ABB RAPID module: 00064353

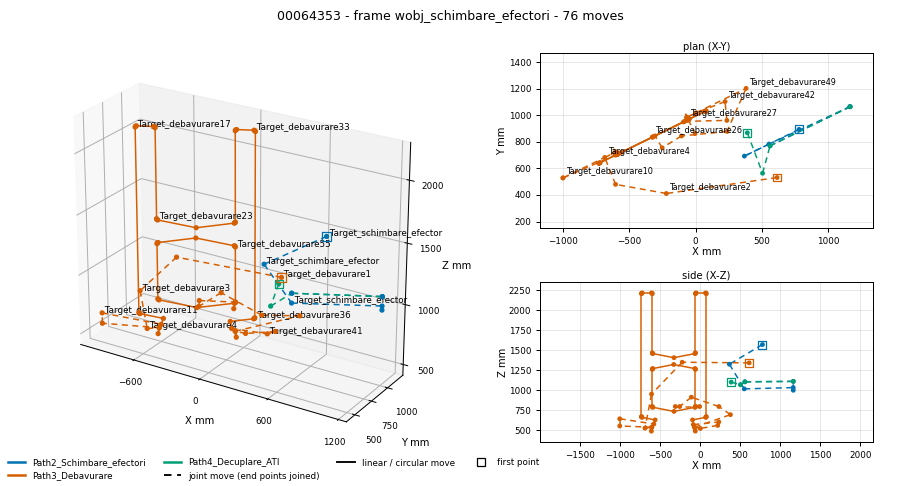
[picture p0: tool path of 00064353 in frame wobj_schimbare_efectori, 76 of 136 moves have a stored position in this frame; points joined in program order, loops and branches not executed]
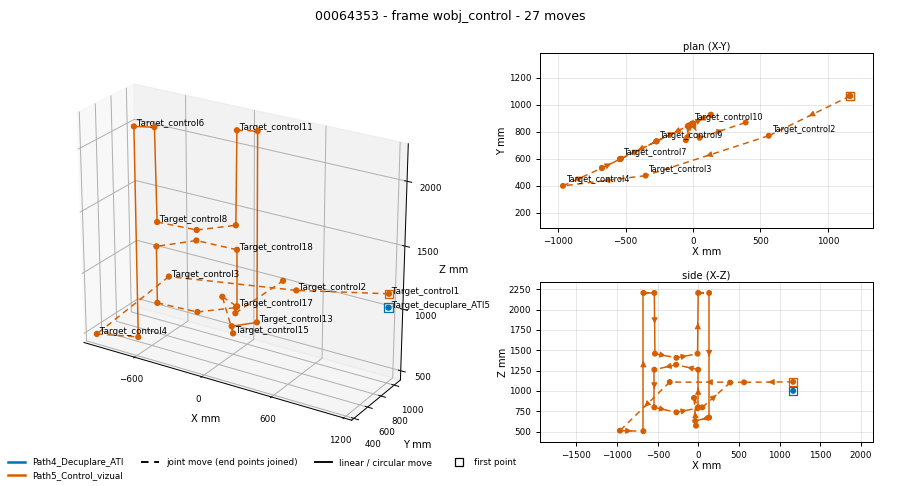
[picture p1: tool path of 00064353 in frame wobj_control, 27 of 136 moves have a stored position in this frame; points joined in program order, loops and branches not executed]
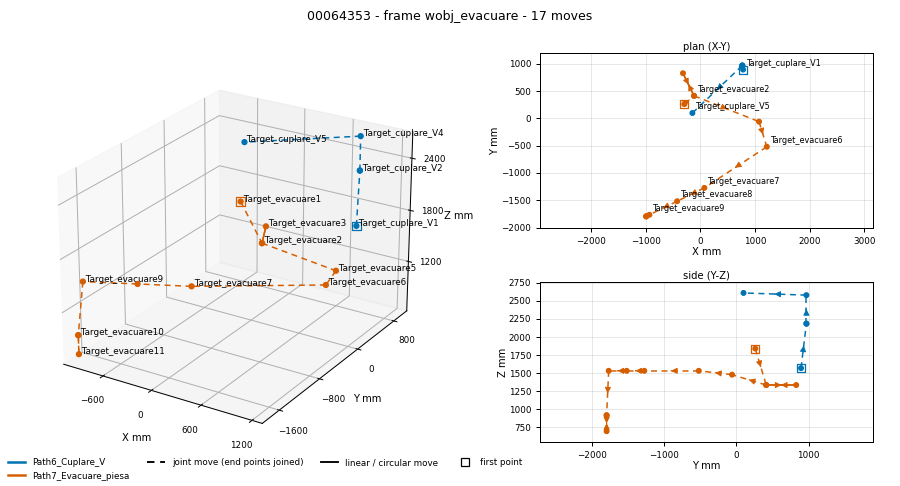
[picture p2: tool path of 00064353 in frame wobj_evacuare, 17 of 136 moves have a stored position in this frame; points joined in program order, loops and branches not executed]
MODULE Module1
	CONST robtarget Target_20_2:=[[0,0.000001,500],[0,0,1,-0.000000001],[-2,-1,0,0],[9E+09,9E+09,9E+09,9E+09,9E+09,9E+09]];
	CONST robtarget Target_10:=[[3.472963553,17.439983187,29.999999981],[0,0,1,-0.000000001],[0,-1,0,0],[9E+09,9E+09,9E+09,9E+09,9E+09,9E+09]];
	CONST robtarget Target_20:=[[0,0.000001,500],[0,0,1,-0.000000001],[-2,-1,0,0],[9E+09,9E+09,9E+09,9E+09,9E+09,9E+09]];
	CONST robtarget Target_20_2_3:=[[493.307337926,-365.839908027,1036.754553389],[0,0,1,-0.000000001],[-1,0,0,0],[9E+09,9E+09,9E+09,9E+09,9E+09,9E+09]];
	CONST robtarget Target_30:=[[-807.278732186,-859.510215676,1233.208067661],[0.579227966,0.405579787,-0.5,-0.5],[0,0,0,0],[9E+09,9E+09,9E+09,9E+09,9E+09,9E+09]];
	CONST robtarget Target_30_3:=[[-1171.792571204,-860.224752875,1298.599208728],[0.579227966,0.405579787,-0.5,-0.5],[1,0,0,0],[9E+09,9E+09,9E+09,9E+09,9E+09,9E+09]];
	CONST robtarget Target_70:=[[-584.684106736,-1037.65235773,1745.210003217],[0.579227966,0.405579787,-0.5,-0.5],[0,0,0,4],[9E+09,9E+09,9E+09,9E+09,9E+09,9E+09]];
	CONST robtarget Target_120:=[[614.35326876,531.541624289,1341.660223262],[0.630196274,-0.425266678,-0.564932078,-0.320706495],[0,0,1,0],[9E+09,9E+09,9E+09,9E+09,9E+09,9E+09]];
	CONST robtarget Target_130:=[[-220.756964436,411.144811502,1349.578986688],[0.630196274,-0.425266678,-0.564932078,-0.320706495],[1,1,0,1],[9E+09,9E+09,9E+09,9E+09,9E+09,9E+09]];
	CONST robtarget Target_140:=[[-603.640790819,480.038707024,951.826023694],[0.630196274,-0.425266678,-0.564932078,-0.320706495],[1,0,1,1],[9E+09,9E+09,9E+09,9E+09,9E+09,9E+09]];
	CONST robtarget Target_150:=[[-684.956865831,682.802213826,527.356838346],[0.630196274,-0.425266678,-0.564932078,-0.320706495],[1,0,1,1],[9E+09,9E+09,9E+09,9E+09,9E+09,9E+09]];
	CONST robtarget Target_160:=[[-600.231193595,724.230019574,538.596152517],[0.630196274,-0.425266678,-0.564932078,-0.320706495],[1,0,1,1],[9E+09,9E+09,9E+09,9E+09,9E+09,9E+09]];
	CONST robtarget Target_170:=[[-615.502782618,744.38841834,511.008322261],[0.630196274,-0.425266678,-0.564932078,-0.320706495],[1,0,1,1],[9E+09,9E+09,9E+09,9E+09,9E+09,9E+09]];
	CONST robtarget Target_180:=[[-605.289704553,715.096779867,490.071182954],[0.630196274,-0.425266678,-0.564932078,-0.320706495],[1,0,1,1],[9E+09,9E+09,9E+09,9E+09,9E+09,9E+09]];
	CONST robtarget Target_190:=[[-592.759513668,700.25774586,516.943595123],[0.630196274,-0.425266678,-0.564932078,-0.320706495],[1,0,1,1],[9E+09,9E+09,9E+09,9E+09,9E+09,9E+09]];
	CONST robtarget Target_200:=[[-600.231193595,724.230019574,538.596152517],[0.630196274,-0.425266678,-0.564932078,-0.320706495],[1,0,1,1],[9E+09,9E+09,9E+09,9E+09,9E+09,9E+09]];
	CONST robtarget Target_210:=[[-1000.069986007,528.723234139,554.74513186],[0.630196274,-0.425266678,-0.564932078,-0.320706495],[1,0,1,1],[9E+09,9E+09,9E+09,9E+09,9E+09,9E+09]];
	CONST robtarget Target_210_2:=[[-1000.069986007,528.723234139,644.473462045],[0.74632501,0.144907108,-0.626241041,0.172693565],[1,-1,2,1],[9E+09,9E+09,9E+09,9E+09,9E+09,9E+09]];
	CONST robtarget Target_220:=[[-574.244255672,714.673851005,578.901883612],[0.74632501,0.144907108,-0.626241041,0.172693565],[1,-2,-2,1],[9E+09,9E+09,9E+09,9E+09,9E+09,9E+09]];
	CONST robtarget Target_230:=[[-558.661492442,722.293261641,630.386873665],[0.74632501,0.144907108,-0.626241041,0.172693565],[1,-2,-2,1],[9E+09,9E+09,9E+09,9E+09,9E+09,9E+09]];
	CONST robtarget Target_240:=[[-721.925864829,642.46285692,662.431918782],[0.74632501,0.144907108,-0.626241041,0.172693565],[1,-1,-2,1],[9E+09,9E+09,9E+09,9E+09,9E+09,9E+09]];
	CONST robtarget Target_250:=[[-727.247702444,639.860669777,665.852120215],[0.74632501,0.144907108,-0.626241041,0.172693565],[1,-1,-2,1],[9E+09,9E+09,9E+09,9E+09,9E+09,9E+09]];
	CONST robtarget Target_260:=[[-729.349460263,638.832985813,672.279996312],[0.74632501,0.144907108,-0.626241041,0.172693565],[1,-1,-2,1],[9E+09,9E+09,9E+09,9E+09,9E+09,9E+09]];
	CONST robtarget Target_270:=[[-729.349460263,638.832985813,2203.889],[0.74632501,0.144907108,-0.626241041,0.172693565],[1,-1,-1,1],[9E+09,9E+09,9E+09,9E+09,9E+09,9E+09]];
	CONST robtarget Target_280:=[[-726.718231405,640.119562068,2210.960067812],[0.74632501,0.144907108,-0.626241041,0.172693565],[1,-1,-1,1],[9E+09,9E+09,9E+09,9E+09,9E+09,9E+09]];
	CONST robtarget Target_290:=[[-720.36588301,643.22563191,2213.889],[0.970550763,-0.019647992,0.084912189,0.22457759],[1,0,-2,1],[9E+09,9E+09,9E+09,9E+09,9E+09,9E+09]];
	CONST robtarget Target_300:=[[-603.579378711,700.33003116,2213.889],[0.970550763,-0.019647992,0.084912189,0.22457759],[1,0,-2,1],[9E+09,9E+09,9E+09,9E+09,9E+09,9E+09]];
	CONST robtarget Target_310:=[[-597.227030315,703.436101002,2210.960067812],[0.970550763,-0.019647992,0.084912189,0.22457759],[1,0,-2,1],[9E+09,9E+09,9E+09,9E+09,9E+09,9E+09]];
	CONST robtarget Target_320:=[[-594.595801457,704.722677256,2203.889],[0.970550763,-0.019647992,0.084912189,0.22457759],[1,0,-2,1],[9E+09,9E+09,9E+09,9E+09,9E+09,9E+09]];
	CONST robtarget Target_330:=[[-594.595801457,704.722677256,1467.279996312],[0.970550763,-0.019647992,0.084912189,0.22457759],[1,0,-2,1],[9E+09,9E+09,9E+09,9E+09,9E+09,9E+09]];
	CONST robtarget Target_340:=[[-592.494043638,705.75036122,1460.852120215],[0.970550763,-0.019647992,0.084912189,0.22457759],[1,0,-2,1],[9E+09,9E+09,9E+09,9E+09,9E+09,9E+09]];
	CONST robtarget Target_350:=[[-587.172206023,708.352548362,1457.431918782],[0.970550763,-0.019647992,0.084912189,0.22457759],[1,0,-2,1],[9E+09,9E+09,9E+09,9E+09,9E+09,9E+09]];
	CONST robtarget Target_360:=[[-323.528502026,837.264835131,1406.297094376],[0.970550763,-0.019647992,0.084912189,0.22457759],[1,0,-1,1],[9E+09,9E+09,9E+09,9E+09,9E+09,9E+09]];
	CONST robtarget Target_370:=[[-63.004761668,964.65157192,1457.431918782],[0.970550763,-0.019647992,0.084912189,0.22457759],[1,0,-1,1],[9E+09,9E+09,9E+09,9E+09,9E+09,9E+09]];
	CONST robtarget Target_380:=[[-57.682924053,967.253759063,1460.852120215],[0.970550763,-0.019647992,0.084912189,0.22457759],[1,0,-1,1],[9E+09,9E+09,9E+09,9E+09,9E+09,9E+09]];
	CONST robtarget Target_390:=[[-55.581166233,968.281443027,1467.279996312],[0.970550763,-0.019647992,0.084912189,0.22457759],[1,0,-1,1],[9E+09,9E+09,9E+09,9E+09,9E+09,9E+09]];
	CONST robtarget Target_400:=[[-55.581166233,968.281443027,2203.889],[0.970550763,-0.019647992,0.084912189,0.22457759],[1,0,-1,1],[9E+09,9E+09,9E+09,9E+09,9E+09,9E+09]];
	CONST robtarget Target_410:=[[-52.949937375,969.568019281,2210.960067812],[0.970550763,-0.019647992,0.084912189,0.22457759],[1,0,-1,1],[9E+09,9E+09,9E+09,9E+09,9E+09,9E+09]];
	CONST robtarget Target_420:=[[-46.59758898,972.674089123,2213.889],[0.970550763,-0.019647992,0.084912189,0.22457759],[1,0,-1,1],[9E+09,9E+09,9E+09,9E+09,9E+09,9E+09]];
	CONST robtarget Target_430:=[[70.188915319,1029.778488373,2213.889],[0.970550763,-0.019647992,0.084912189,0.22457759],[0,0,-1,1],[9E+09,9E+09,9E+09,9E+09,9E+09,9E+09]];
	CONST robtarget Target_440:=[[76.541263714,1032.884558215,2210.960067812],[0.970550763,-0.019647992,0.084912189,0.22457759],[0,0,-1,1],[9E+09,9E+09,9E+09,9E+09,9E+09,9E+09]];
	CONST robtarget Target_450:=[[79.172492573,1034.171134469,2203.889],[0.626241041,-0.172693565,0.74632501,0.144907108],[1,1,-2,1],[9E+09,9E+09,9E+09,9E+09,9E+09,9E+09]];
	CONST robtarget Target_460:=[[79.172492573,1034.171134469,672.279996312],[0.626241041,-0.172693565,0.74632501,0.144907108],[1,0,-1,1],[9E+09,9E+09,9E+09,9E+09,9E+09,9E+09]];
	CONST robtarget Target_470:=[[77.070734753,1033.143450506,665.852120215],[0.626241041,-0.172693565,0.74632501,0.144907108],[1,0,-1,1],[9E+09,9E+09,9E+09,9E+09,9E+09,9E+09]];
	CONST robtarget Target_480:=[[71.748897138,1030.541263363,662.431918782],[0.626241041,-0.172693565,0.74632501,0.144907108],[1,0,-1,1],[9E+09,9E+09,9E+09,9E+09,9E+09,9E+09]];
	CONST robtarget Target_490:=[[-91.515475248,950.710858642,630.386873665],[0.626241041,-0.172693565,0.74632501,0.144907108],[1,1,-1,1],[9E+09,9E+09,9E+09,9E+09,9E+09,9E+09]];
	CONST robtarget Target_500:=[[-82.17325952,955.27886605,571.409990938],[0.626241041,-0.172693565,0.74632501,0.144907108],[1,1,-1,1],[9E+09,9E+09,9E+09,9E+09,9E+09,9E+09]];
	CONST robtarget Target_500_2:=[[235.647161917,962.336296138,604.766182313],[0.626241041,-0.172693565,0.74632501,0.144907108],[0,0,-1,1],[9E+09,9E+09,9E+09,9E+09,9E+09,9E+09]];
	CONST robtarget Target_500_2_2:=[[222.398190082,1104.203348059,561.899220237],[0.320706496,-0.564932078,0.425266677,0.630196274],[0,1,-2,0],[9E+09,9E+09,9E+09,9E+09,9E+09,9E+09]];
	CONST robtarget Target_510:=[[4.592265391,1019.966932715,523.466438018],[0.425266678,-0.630196274,0.320706495,0.564932078],[0,1,-2,0],[9E+09,9E+09,9E+09,9E+09,9E+09,9E+09]];
	CONST robtarget Target_520:=[[-67.51635848,984.708409724,538.596152517],[0.425266678,-0.630196274,0.320706495,0.564932078],[0,1,-2,0],[9E+09,9E+09,9E+09,9E+09,9E+09,9E+09]];
	CONST robtarget Target_530:=[[-74.04786326,1009.140395264,511.008322261],[0.425266678,-0.630196274,0.320706495,0.564932078],[0,1,-2,0],[9E+09,9E+09,9E+09,9E+09,9E+09,9E+09]];
	CONST robtarget Target_540:=[[-57.20170243,983.09209564,490.071182954],[0.425266678,-0.630196274,0.320706495,0.564932078],[0,1,-2,0],[9E+09,9E+09,9E+09,9E+09,9E+09,9E+09]];
	CONST robtarget Target_550:=[[-53.184944606,964.090299134,516.943595123],[0.425266678,-0.630196274,0.320706495,0.564932078],[0,1,-2,0],[9E+09,9E+09,9E+09,9E+09,9E+09,9E+09]];
	CONST robtarget Target_560:=[[-67.51635848,984.708409724,538.596152517],[0.425266678,-0.630196274,0.320706495,0.564932078],[0,1,-2,0],[9E+09,9E+09,9E+09,9E+09,9E+09,9E+09]];
	CONST robtarget Target_570:=[[380.563228786,1203.803208398,695.774665043],[0.425266678,-0.630196274,0.320706495,0.564932078],[0,1,-2,0],[9E+09,9E+09,9E+09,9E+09,9E+09,9E+09]];
	CONST robtarget Target_580_3:=[[236.855316057,878.977367128,797.279996312],[0.626241041,-0.172693565,0.74632501,0.144907108],[0,0,-1,1],[9E+09,9E+09,9E+09,9E+09,9E+09,9E+09]];
	CONST robtarget Target_740:=[[-106.574951523,844.917671275,913.754533399],[0.626241041,-0.172693565,0.74632501,0.144907108],[1,1,-1,1],[9E+09,9E+09,9E+09,9E+09,9E+09,9E+09]];
	CONST robtarget Target_580_3_2:=[[-251.957733199,755.881530829,797.279996312],[0.626241041,-0.172693565,0.74632501,0.144907108],[1,1,-1,1],[9E+09,9E+09,9E+09,9E+09,9E+09,9E+09]];
	CONST robtarget Target_580:=[[-306.602704629,845.540941159,797.279996312],[0.626241041,-0.172693565,0.74632501,0.144907108],[1,1,-1,1],[9E+09,9E+09,9E+09,9E+09,9E+09,9E+09]];
	CONST robtarget Target_590:=[[-55.581166233,968.281443027,797.279996312],[0.626241041,-0.172693565,0.74632501,0.144907108],[1,1,-1,1],[9E+09,9E+09,9E+09,9E+09,9E+09,9E+09]];
	CONST robtarget Target_600:=[[-55.581166233,968.281443027,1260.498003688],[0.626241041,-0.172693565,0.74632501,0.144907108],[1,1,-1,1],[9E+09,9E+09,9E+09,9E+09,9E+09,9E+09]];
	CONST robtarget Target_610:=[[-57.682924053,967.253759063,1266.925879785],[0.626241041,-0.172693565,0.74632501,0.144907108],[1,1,-1,1],[9E+09,9E+09,9E+09,9E+09,9E+09,9E+09]];
	CONST robtarget Target_620:=[[-63.004761668,964.65157192,1270.346081218],[0.626241041,-0.172693565,0.74632501,0.144907108],[1,1,-1,1],[9E+09,9E+09,9E+09,9E+09,9E+09,9E+09]];
	CONST robtarget Target_630:=[[-326.648465665,835.739285151,1321.480905624],[0.626241041,-0.172693565,0.74632501,0.144907108],[1,1,-1,1],[9E+09,9E+09,9E+09,9E+09,9E+09,9E+09]];
	CONST robtarget Target_640:=[[-587.172206023,708.352548362,1270.346081218],[0.626241041,-0.172693565,0.74632501,0.144907108],[1,1,-1,1],[9E+09,9E+09,9E+09,9E+09,9E+09,9E+09]];
	CONST robtarget Target_650:=[[-592.494043638,705.75036122,1266.925879785],[0.626241041,-0.172693565,0.74632501,0.144907108],[1,1,-1,1],[9E+09,9E+09,9E+09,9E+09,9E+09,9E+09]];
	CONST robtarget Target_660:=[[-594.595801457,704.722677256,1260.498003688],[0.626241041,-0.172693565,0.74632501,0.144907108],[1,1,-1,1],[9E+09,9E+09,9E+09,9E+09,9E+09,9E+09]];
	CONST robtarget Target_670:=[[-594.595801457,704.722677256,797.279996312],[0.626241041,-0.172693565,0.74632501,0.144907108],[1,1,-1,1],[9E+09,9E+09,9E+09,9E+09,9E+09,9E+09]];
	CONST robtarget Target_680:=[[-592.494043638,705.75036122,790.852120215],[0.626241041,-0.172693565,0.74632501,0.144907108],[1,1,-1,1],[9E+09,9E+09,9E+09,9E+09,9E+09,9E+09]];
	CONST robtarget Target_690:=[[-587.172206023,708.352548362,787.431918782],[0.626241041,-0.172693565,0.74632501,0.144907108],[1,1,-1,1],[9E+09,9E+09,9E+09,9E+09,9E+09,9E+09]];
	CONST robtarget Target_700:=[[-323.528502026,837.264835131,736.297094376],[0.626241041,-0.172693565,0.74632501,0.144907108],[1,1,-1,1],[9E+09,9E+09,9E+09,9E+09,9E+09,9E+09]];
	CONST robtarget Target_710:=[[-63.004761668,964.65157192,787.431918782],[0.626241041,-0.172693565,0.74632501,0.144907108],[1,1,-1,1],[9E+09,9E+09,9E+09,9E+09,9E+09,9E+09]];
	CONST robtarget Target_720:=[[-57.682924053,967.253759063,790.852120215],[0.626241041,-0.172693565,0.74632501,0.144907108],[1,1,-1,1],[9E+09,9E+09,9E+09,9E+09,9E+09,9E+09]];
	CONST robtarget Target_730:=[[-55.581166233,968.281443027,797.279996312],[0.626241041,-0.172693565,0.74632501,0.144907108],[1,1,-1,1],[9E+09,9E+09,9E+09,9E+09,9E+09,9E+09]];
	CONST robtarget Target_730_2:=[[-4.129380996,863.055327059,797.279996312],[0.626241041,-0.172693565,0.74632501,0.144907108],[1,1,-1,1],[9E+09,9E+09,9E+09,9E+09,9E+09,9E+09]];
	CONST robtarget Target_750:=[[353.286050265,-1090.926157105,1000],[0,0,1,-0.000000001],[-1,0,-1,0],[9E+09,9E+09,9E+09,9E+09,9E+09,9E+09]];
	CONST robtarget Target_100_2:=[[1164.241304795,1065.453076327,1110.91287582],[0,0.848311443,-0.529497588,0],[0,0,-1,0],[9E+09,9E+09,9E+09,9E+09,9E+09,9E+09]];
	CONST robtarget Target_110_3:=[[561.343174474,770.657579762,1105.422922565],[0,0.848311443,-0.529497588,0],[0,0,-1,0],[9E+09,9E+09,9E+09,9E+09,9E+09,9E+09]];
	CONST robtarget Target_120_3:=[[-352.181570531,474.725664361,1108.429867517],[0.630196274,-0.425266678,-0.564932078,-0.320706495],[1,-2,-1,0],[9E+09,9E+09,9E+09,9E+09,9E+09,9E+09]];
	CONST robtarget Target_130_3:=[[-965.595492909,398.655755176,510.210088752],[0.630196274,-0.425266678,-0.564932078,-0.320706495],[1,-2,-1,0],[9E+09,9E+09,9E+09,9E+09,9E+09,9E+09]];
	CONST robtarget Target_260_2:=[[-676.765426106,531.291262028,504.173173014],[0.630196274,-0.425266678,-0.564932078,-0.320706495],[1,-2,-1,0],[9E+09,9E+09,9E+09,9E+09,9E+09,9E+09]];
	CONST robtarget Target_270_2:=[[-676.765426106,531.291262028,2203.889],[0.630196274,-0.425266678,-0.564932078,-0.320706495],[1,-1,-2,0],[9E+09,9E+09,9E+09,9E+09,9E+09,9E+09]];
	CONST robtarget Target_320_2:=[[-542.0117673,597.180953471,2203.889],[0.630196274,-0.425266678,-0.564932078,-0.320706495],[1,-1,-2,0],[9E+09,9E+09,9E+09,9E+09,9E+09,9E+09]];
	CONST robtarget Target_350_2:=[[-534.588171866,600.810824577,1457.431918782],[0.630196274,-0.425266678,-0.564932078,-0.320706495],[1,-1,-1,0],[9E+09,9E+09,9E+09,9E+09,9E+09,9E+09]];
	CONST robtarget Target_360_2:=[[-270.944467869,729.723111346,1406.297094376],[0.630196274,-0.425266678,-0.564932078,-0.320706495],[1,-1,-1,1],[9E+09,9E+09,9E+09,9E+09,9E+09,9E+09]];
	CONST robtarget Target_370_2:=[[-10.420727511,857.109848135,1457.431918782],[0.630196274,-0.425266678,-0.564932078,-0.320706495],[0,-1,-1,1],[9E+09,9E+09,9E+09,9E+09,9E+09,9E+09]];
	CONST robtarget Target_400_2:=[[-2.997132076,860.739719242,2203.889],[0.630196274,-0.425266678,-0.564932078,-0.320706495],[0,-2,-1,1],[9E+09,9E+09,9E+09,9E+09,9E+09,9E+09]];
	CONST robtarget Target_450_2:=[[131.75652673,926.629410684,2203.889],[0.630196274,-0.425266678,-0.564932078,-0.320706495],[0,-2,-1,1],[9E+09,9E+09,9E+09,9E+09,9E+09,9E+09]];
	CONST robtarget Target_460_2:=[[131.75652673,926.629410684,672.279996312],[0.630196274,-0.425266678,-0.564932078,-0.320706495],[0,-1,-2,1],[9E+09,9E+09,9E+09,9E+09,9E+09,9E+09]];
	CONST robtarget Target_490_2:=[[-38.931441091,843.169134857,630.386873665],[0.630196274,-0.425266678,-0.564932078,-0.320706495],[0,-1,-2,1],[9E+09,9E+09,9E+09,9E+09,9E+09,9E+09]];
	CONST robtarget Target_500_3:=[[-29.589225363,847.737142265,571.409990938],[0.630196274,-0.425266678,-0.564932078,-0.320706495],[0,-1,-2,1],[9E+09,9E+09,9E+09,9E+09,9E+09,9E+09]];
	CONST robtarget Target_740_2:=[[-53.990917366,737.37594749,913.754533399],[0.630196274,-0.425266678,-0.564932078,-0.320706495],[0,-1,-2,1],[9E+09,9E+09,9E+09,9E+09,9E+09,9E+09]];
	CONST robtarget Target_590_2:=[[-2.997132076,860.739719242,797.279996312],[0.630196274,-0.425266678,-0.564932078,-0.320706495],[0,-1,-2,1],[9E+09,9E+09,9E+09,9E+09,9E+09,9E+09]];
	CONST robtarget Target_600_2:=[[-2.997132076,860.739719242,1260.498003688],[0.630196274,-0.425266678,-0.564932078,-0.320706495],[0,-1,-2,1],[9E+09,9E+09,9E+09,9E+09,9E+09,9E+09]];
	CONST robtarget Target_630_2:=[[-274.064431508,728.197561366,1321.480905624],[0.630196274,-0.425266678,-0.564932078,-0.320706495],[1,-1,-2,1],[9E+09,9E+09,9E+09,9E+09,9E+09,9E+09]];
	CONST robtarget Target_660_2:=[[-542.0117673,597.180953471,1260.498003688],[0.630196274,-0.425266678,-0.564932078,-0.320706495],[1,-2,-1,0],[9E+09,9E+09,9E+09,9E+09,9E+09,9E+09]];
	CONST robtarget Target_670_2:=[[-542.0117673,597.180953471,797.279996312],[0.630196274,-0.425266678,-0.564932078,-0.320706495],[1,-2,-1,0],[9E+09,9E+09,9E+09,9E+09,9E+09,9E+09]];
	CONST robtarget Target_700_2:=[[-270.944467869,729.723111346,736.297094376],[0.630196274,-0.425266678,-0.564932078,-0.320706495],[1,-1,-2,1],[9E+09,9E+09,9E+09,9E+09,9E+09,9E+09]];
	CONST robtarget Target_710_2:=[[-10.420727511,857.109848135,787.431918782],[0.630196274,-0.425266678,-0.564932078,-0.320706495],[0,-1,-2,1],[9E+09,9E+09,9E+09,9E+09,9E+09,9E+09]];
	CONST robtarget Target_730_3:=[[-2.997132076,860.739719242,797.279996312],[0.630196274,-0.425266678,-0.564932078,-0.320706495],[0,-1,-2,1],[9E+09,9E+09,9E+09,9E+09,9E+09,9E+09]];
	CONST robtarget Target_730_2_2:=[[48.454653161,755.513603274,797.279996312],[0.630196274,-0.425266678,-0.564932078,-0.320706495],[0,-1,-2,1],[9E+09,9E+09,9E+09,9E+09,9E+09,9E+09]];
	CONST robtarget Target_130_2_2:=[[389.997020927,869.040623857,1101.572770211],[0.630196274,-0.425266678,-0.564932078,-0.320706495],[0,-1,-2,1],[9E+09,9E+09,9E+09,9E+09,9E+09,9E+09]];
	CONST robtarget Target_80_2_2:=[[-148.366452112,98.986292765,2610.344805667],[0.159406928,0.159406928,-0.688904515,-0.688904516],[1,0,0,4],[9E+09,9E+09,9E+09,9E+09,9E+09,9E+09]];
	CONST robtarget Target_70_2:=[[-297.408117168,261.539979913,1840.929204997],[0.159406928,0.159406928,-0.688904515,-0.688904516],[0,0,0,4],[9E+09,9E+09,9E+09,9E+09,9E+09,9E+09]];
	CONST robtarget Target_30_2:=[[-117.985307131,412.947477324,1336.176966578],[0.159406928,0.159406928,-0.688904515,-0.688904516],[0,0,0,0],[9E+09,9E+09,9E+09,9E+09,9E+09,9E+09]];
	CONST robtarget Target_30_3_2:=[[-320.695795916,827.518853271,1336.176966578],[0.159406928,0.159406928,-0.688904515,-0.688904516],[1,0,0,0],[9E+09,9E+09,9E+09,9E+09,9E+09,9E+09]];
	CONST robtarget Target_30_2_2:=[[-117.985307131,412.947477324,1336.176966578],[0.159406928,0.159406928,-0.688904515,-0.688904516],[0,0,0,0],[9E+09,9E+09,9E+09,9E+09,9E+09,9E+09]];
	CONST robtarget Target_30_2_3:=[[1072.781898944,-59.825918958,1479.636846222],[0.374411334,0.374411335,0.599846774,0.599846775],[-1,1,-1,0],[9E+09,9E+09,9E+09,9E+09,9E+09,9E+09]];
	CONST robtarget Target_30_2_3_2:=[[1215.425844801,-519.48484737,1533.087792477],[0.374411334,0.374411335,0.599846774,0.599846775],[-1,1,-1,0],[9E+09,9E+09,9E+09,9E+09,9E+09,9E+09]];
	CONST robtarget Target_30_2_3_2_2:=[[71.368530681,-1273.53877769,1533.087792477],[0.688904515,0.688904516,0.159406928,0.159406928],[-2,1,-1,0],[9E+09,9E+09,9E+09,9E+09,9E+09,9E+09]];
	CONST robtarget Target_30_2_3_2_2_2:=[[-427.431513587,-1517.434055188,1533.087792477],[0.000000001,0.974258109,0.225435439,0],[-2,-1,0,0],[9E+09,9E+09,9E+09,9E+09,9E+09,9E+09]];
	CONST robtarget Target_30_2_3_2_2_2_2:=[[-935.838539063,-1766.02680089,1533.087792477],[-0.000000001,0.974258109,0.225435439,0],[-2,0,0,0],[9E+09,9E+09,9E+09,9E+09,9E+09,9E+09]];
	CONST robtarget Target_30_2_3_2_2_2_2_2:=[[-994.92710219,-1794.918982569,917.887564527],[0.000000001,0.974258109,0.225435439,0],[-2,-1,0,0],[9E+09,9E+09,9E+09,9E+09,9E+09,9E+09]];
	CONST robtarget Target_30_2_3_2_2_2_2_2_2:=[[-994.92710219,-1794.918982569,697.821327506],[-0.000000001,0.974258109,0.225435439,0],[-2,0,0,0],[9E+09,9E+09,9E+09,9E+09,9E+09,9E+09]];
	CONST robtarget Target_130_2:=[[389.997020927,869.040623857,1101.572770211],[0.630196274,-0.425266678,-0.564932078,-0.320706495],[0,1,0,0],[9E+09,9E+09,9E+09,9E+09,9E+09,9E+09]];
	CONST robtarget Target_120_2:=[[504.928038476,563.849286682,1069.091100494],[0,0.848311443,-0.529497588,0],[0,0,-1,0],[9E+09,9E+09,9E+09,9E+09,9E+09,9E+09]];
	CONST robtarget Target_110_2:=[[561.343174474,770.657579762,1105.422922565],[0,0.848311443,-0.529497588,0],[0,0,-1,0],[9E+09,9E+09,9E+09,9E+09,9E+09,9E+09]];
	CONST robtarget Target_100:=[[1164.241304795,1065.453076327,1110.91287582],[0,0.848311443,-0.529497588,0],[0,0,-1,0],[9E+09,9E+09,9E+09,9E+09,9E+09,9E+09]];
	CONST robtarget Target_90_2_2_3_2_2_2_2:=[[1164.456250233,1065.58489233,1000],[0,0.848311443,-0.529497588,0],[0,0,-1,0],[9E+09,9E+09,9E+09,9E+09,9E+09,9E+09]];
	CONST robtarget Target_80_2:=[[-176.063589295,-890.179717053,2221.711117045],[0.579227966,0.405579787,-0.5,-0.5],[1,0,0,4],[9E+09,9E+09,9E+09,9E+09,9E+09,9E+09]];
	CONST robtarget Target_80:=[[-549.798887424,-878.736368632,2286.609570489],[0.69636424,-0.122787804,0,-0.707106781],[1,-1,0,1],[9E+09,9E+09,9E+09,9E+09,9E+09,9E+09]];
	CONST robtarget Target_90:=[[-658.456780387,304.505009965,2066.113793534],[0.69636424,-0.122787804,0,-0.707106781],[0,-1,1,1],[9E+09,9E+09,9E+09,9E+09,9E+09,9E+09]];
	CONST robtarget Target_90_2:=[[-690.279328221,273.165917946,1888.380971862],[0.69636424,-0.122787804,0,-0.707106781],[0,-1,1,1],[9E+09,9E+09,9E+09,9E+09,9E+09,9E+09]];
	CONST robtarget Target_90_2_2:=[[779.908229606,894.538776646,1570.162539077],[0.225435439,0,0,-0.974258109],[0,0,1,1],[9E+09,9E+09,9E+09,9E+09,9E+09,9E+09]];
	CONST robtarget Target_90_2_2_3:=[[367.891360431,693.077349856,1324.929850073],[0,0.848311443,-0.529497588,0],[0,0,-1,0],[9E+09,9E+09,9E+09,9E+09,9E+09,9E+09]];
	CONST robtarget Target_90_2_2_3_2:=[[553.518951213,783.842563864,1017.503826288],[0,0.848311443,-0.529497588,0],[0,0,-1,0],[9E+09,9E+09,9E+09,9E+09,9E+09,9E+09]];
	CONST robtarget Target_90_2_2_3_2_2:=[[1164.456250233,1065.58489233,1033.237043133],[0,0.848311443,-0.529497588,0],[0,0,-1,0],[9E+09,9E+09,9E+09,9E+09,9E+09,9E+09]];
	CONST robtarget Target_90_2_2_3_2_2_2:=[[1164.456250233,1065.58489233,1000],[0,0.848311443,-0.529497588,0],[0,0,-1,0],[9E+09,9E+09,9E+09,9E+09,9E+09,9E+09]];
	CONST robtarget Target_110:=[[561.343174474,770.657579762,1105.422922565],[0,0.848311443,-0.529497588,0],[0,0,-1,0],[9E+09,9E+09,9E+09,9E+09,9E+09,9E+09]];
	CONST robtarget Target_80_3:=[[-315.067708607,439.913739054,2610.344805668],[0.225435439,0,0,-0.974258109],[1,0,0,1],[9E+09,9E+09,9E+09,9E+09,9E+09,9E+09]];
	CONST robtarget Target_130_2_2_2:=[[389.997020927,869.040623857,1101.572770211],[0.630196274,-0.425266678,-0.564932078,-0.320706495],[0,-1,-2,1],[9E+09,9E+09,9E+09,9E+09,9E+09,9E+09]];
	CONST robtarget Target_90_2_2_2:=[[779.908229606,894.538776646,1570.162539077],[0.225435439,0,0,-0.974258109],[0,0,1,1],[9E+09,9E+09,9E+09,9E+09,9E+09,9E+09]];
	CONST robtarget Target_90_2_3:=[[766.154301146,968.592405176,2185.609751442],[0.225435439,0,0,-0.974258109],[0,0,1,1],[9E+09,9E+09,9E+09,9E+09,9E+09,9E+09]];
	CONST robtarget Target_90_2_4:=[[766.154301146,968.592405176,2185.609751442],[0.225435439,0,0,-0.974258109],[0,0,1,1],[9E+09,9E+09,9E+09,9E+09,9E+09,9E+09]];
	CONST robtarget Target_90_3:=[[766.154301147,968.592405175,2579.975738982],[0.225435439,0,0,-0.974258109],[0,0,1,1],[9E+09,9E+09,9E+09,9E+09,9E+09,9E+09]];
	CONST robtarget Target_20_2_3_2:=[[444.870488584,-801.565485803,1694.675220196],[0,0,0.422618263,0.906307786],[-1,1,0,0],[9E+09,9E+09,9E+09,9E+09,9E+09,9E+09]];
	CONST robtarget Target_20_2_3_2_4:=[[-62.368508603,-801.565493431,1694.675207733],[0.346828974,-0.161729008,-0.390448363,-0.837319214],[0,0,0,5],[9E+09,9E+09,9E+09,9E+09,9E+09,9E+09]];
	CONST robtarget Target_preluare_piesa3:=[[0,0.000001,500],[0,0,1,-0.000000001],[-2,-1,0,0],[9E+09,9E+09,9E+09,9E+09,9E+09,9E+09]];
	CONST robtarget Target_preluare_piesa2:=[[3.472963553,17.439983187,29.999999981],[0,0,1,-0.000000001],[0,-1,0,0],[9E+09,9E+09,9E+09,9E+09,9E+09,9E+09]];
	CONST robtarget Target_preluare_piesa1:=[[0,0.000001,500],[0,0,1,-0.000000001],[-2,-1,0,0],[9E+09,9E+09,9E+09,9E+09,9E+09,9E+09]];
	CONST robtarget Target_preluare_piesa4:=[[493.307337926,-365.839908027,1036.754553389],[0,0,1,-0.000000001],[-1,0,0,0],[9E+09,9E+09,9E+09,9E+09,9E+09,9E+09]];
	CONST robtarget Target_preluare_piesa5:=[[444.870488584,-801.565485803,1694.675220196],[0,0,0.422618263,0.906307786],[-1,1,0,0],[9E+09,9E+09,9E+09,9E+09,9E+09,9E+09]];
	CONST robtarget Target_preluare_piesa6:=[[-62.368508603,-801.565493431,1694.675207733],[0.346828974,-0.161729008,-0.390448363,-0.837319214],[0,0,0,5],[9E+09,9E+09,9E+09,9E+09,9E+09,9E+09]];
	CONST robtarget Target_preluare_piesa7:=[[-807.278732186,-859.510215676,1233.208067661],[0.579227966,0.405579787,-0.5,-0.5],[0,0,0,0],[9E+09,9E+09,9E+09,9E+09,9E+09,9E+09]];
	CONST robtarget Target_preluare_piesa8:=[[-1171.792571204,-860.224752875,1298.599208728],[0.579227966,0.405579787,-0.5,-0.5],[1,0,0,0],[9E+09,9E+09,9E+09,9E+09,9E+09,9E+09]];
	CONST robtarget Target_preluare_piesa9:=[[-584.684106736,-1037.65235773,1745.210003217],[0.579227966,0.405579787,-0.5,-0.5],[0,0,0,4],[9E+09,9E+09,9E+09,9E+09,9E+09,9E+09]];
	CONST robtarget Target_debavurare1:=[[614.35326876,531.541624289,1341.660223262],[0.630196274,-0.425266678,-0.564932078,-0.320706495],[0,0,1,0],[9E+09,9E+09,9E+09,9E+09,9E+09,9E+09]];
	CONST robtarget Target_debavurare2:=[[-220.756964436,411.144811502,1349.578986688],[0.630196274,-0.425266678,-0.564932078,-0.320706495],[1,1,0,1],[9E+09,9E+09,9E+09,9E+09,9E+09,9E+09]];
	CONST robtarget Target_debavurare3:=[[-603.640790819,480.038707024,951.826023694],[0.630196274,-0.425266678,-0.564932078,-0.320706495],[1,0,1,1],[9E+09,9E+09,9E+09,9E+09,9E+09,9E+09]];
	CONST robtarget Target_debavurare4:=[[-684.956865831,682.802213826,527.356838346],[0.630196274,-0.425266678,-0.564932078,-0.320706495],[1,0,1,1],[9E+09,9E+09,9E+09,9E+09,9E+09,9E+09]];
	CONST robtarget Target_debavurare5:=[[-600.231193595,724.230019574,538.596152517],[0.630196274,-0.425266678,-0.564932078,-0.320706495],[1,0,1,1],[9E+09,9E+09,9E+09,9E+09,9E+09,9E+09]];
	CONST robtarget Target_debavurare6:=[[-615.502782618,744.38841834,511.008322261],[0.630196274,-0.425266678,-0.564932078,-0.320706495],[1,0,1,1],[9E+09,9E+09,9E+09,9E+09,9E+09,9E+09]];
	CONST robtarget Target_debavurare7:=[[-605.289704553,715.096779867,490.071182954],[0.630196274,-0.425266678,-0.564932078,-0.320706495],[1,0,1,1],[9E+09,9E+09,9E+09,9E+09,9E+09,9E+09]];
	CONST robtarget Target_debavurare8:=[[-592.759513668,700.25774586,516.943595123],[0.630196274,-0.425266678,-0.564932078,-0.320706495],[1,0,1,1],[9E+09,9E+09,9E+09,9E+09,9E+09,9E+09]];
	CONST robtarget Target_debavurare9:=[[-600.231193595,724.230019574,538.596152517],[0.630196274,-0.425266678,-0.564932078,-0.320706495],[1,0,1,1],[9E+09,9E+09,9E+09,9E+09,9E+09,9E+09]];
	CONST robtarget Target_debavurare10:=[[-1000.069986007,528.723234139,554.74513186],[0.630196274,-0.425266678,-0.564932078,-0.320706495],[1,0,1,1],[9E+09,9E+09,9E+09,9E+09,9E+09,9E+09]];
	CONST robtarget Target_debavurare11:=[[-1000.069986007,528.723234139,644.473462045],[0.74632501,0.144907108,-0.626241041,0.172693565],[1,-1,2,1],[9E+09,9E+09,9E+09,9E+09,9E+09,9E+09]];
	CONST robtarget Target_debavurare12:=[[-574.244255672,714.673851005,578.901883612],[0.74632501,0.144907108,-0.626241041,0.172693565],[1,-2,-2,1],[9E+09,9E+09,9E+09,9E+09,9E+09,9E+09]];
	CONST robtarget Target_debavurare13:=[[-558.661492442,722.293261641,630.386873665],[0.74632501,0.144907108,-0.626241041,0.172693565],[1,-2,-2,1],[9E+09,9E+09,9E+09,9E+09,9E+09,9E+09]];
	CONST robtarget Target_debavurare14:=[[-721.925864829,642.46285692,662.431918782],[0.74632501,0.144907108,-0.626241041,0.172693565],[1,-1,-2,1],[9E+09,9E+09,9E+09,9E+09,9E+09,9E+09]];
	CONST robtarget Target_debavurare15:=[[-727.247702444,639.860669777,665.852120215],[0.74632501,0.144907108,-0.626241041,0.172693565],[1,-1,-2,1],[9E+09,9E+09,9E+09,9E+09,9E+09,9E+09]];
	CONST robtarget Target_debavurare16:=[[-729.349460263,638.832985813,672.279996312],[0.74632501,0.144907108,-0.626241041,0.172693565],[1,-1,-2,1],[9E+09,9E+09,9E+09,9E+09,9E+09,9E+09]];
	CONST robtarget Target_debavurare17:=[[-729.349460263,638.832985813,2203.889],[0.74632501,0.144907108,-0.626241041,0.172693565],[1,-1,-1,1],[9E+09,9E+09,9E+09,9E+09,9E+09,9E+09]];
	CONST robtarget Target_debavurare18:=[[-726.718231405,640.119562068,2210.960067812],[0.74632501,0.144907108,-0.626241041,0.172693565],[1,-1,-1,1],[9E+09,9E+09,9E+09,9E+09,9E+09,9E+09]];
	CONST robtarget Target_debavurare19:=[[-720.36588301,643.22563191,2213.889],[0.970550763,-0.019647992,0.084912189,0.22457759],[1,0,-2,1],[9E+09,9E+09,9E+09,9E+09,9E+09,9E+09]];
	CONST robtarget Target_debavurare20:=[[-603.579378711,700.33003116,2213.889],[0.970550763,-0.019647992,0.084912189,0.22457759],[1,0,-2,1],[9E+09,9E+09,9E+09,9E+09,9E+09,9E+09]];
	CONST robtarget Target_debavurare21:=[[-597.227030315,703.436101002,2210.960067812],[0.970550763,-0.019647992,0.084912189,0.22457759],[1,0,-2,1],[9E+09,9E+09,9E+09,9E+09,9E+09,9E+09]];
	CONST robtarget Target_debavurare22:=[[-594.595801457,704.722677256,2203.889],[0.970550763,-0.019647992,0.084912189,0.22457759],[1,0,-2,1],[9E+09,9E+09,9E+09,9E+09,9E+09,9E+09]];
	CONST robtarget Target_debavurare23:=[[-594.595801457,704.722677256,1467.279996312],[0.970550763,-0.019647992,0.084912189,0.22457759],[1,0,-2,1],[9E+09,9E+09,9E+09,9E+09,9E+09,9E+09]];
	CONST robtarget Target_debavurare24:=[[-592.494043638,705.75036122,1460.852120215],[0.970550763,-0.019647992,0.084912189,0.22457759],[1,0,-2,1],[9E+09,9E+09,9E+09,9E+09,9E+09,9E+09]];
	CONST robtarget Target_debavurare25:=[[-587.172206023,708.352548362,1457.431918782],[0.970550763,-0.019647992,0.084912189,0.22457759],[1,0,-2,1],[9E+09,9E+09,9E+09,9E+09,9E+09,9E+09]];
	CONST robtarget Target_debavurare26:=[[-323.528502026,837.264835131,1406.297094376],[0.970550763,-0.019647992,0.084912189,0.22457759],[1,0,-1,1],[9E+09,9E+09,9E+09,9E+09,9E+09,9E+09]];
	CONST robtarget Target_debavurare27:=[[-63.004761668,964.65157192,1457.431918782],[0.970550763,-0.019647992,0.084912189,0.22457759],[1,0,-1,1],[9E+09,9E+09,9E+09,9E+09,9E+09,9E+09]];
	CONST robtarget Target_debavurare28:=[[-57.682924053,967.253759063,1460.852120215],[0.970550763,-0.019647992,0.084912189,0.22457759],[1,0,-1,1],[9E+09,9E+09,9E+09,9E+09,9E+09,9E+09]];
	CONST robtarget Target_debavurare29:=[[-55.581166233,968.281443027,1467.279996312],[0.970550763,-0.019647992,0.084912189,0.22457759],[1,0,-1,1],[9E+09,9E+09,9E+09,9E+09,9E+09,9E+09]];
	CONST robtarget Target_debavurare30:=[[-55.581166233,968.281443027,2203.889],[0.970550763,-0.019647992,0.084912189,0.22457759],[1,0,-1,1],[9E+09,9E+09,9E+09,9E+09,9E+09,9E+09]];
	CONST robtarget Target_debavurare31:=[[-52.949937375,969.568019281,2210.960067812],[0.970550763,-0.019647992,0.084912189,0.22457759],[1,0,-1,1],[9E+09,9E+09,9E+09,9E+09,9E+09,9E+09]];
	CONST robtarget Target_debavurare32:=[[-46.59758898,972.674089123,2213.889],[0.970550763,-0.019647992,0.084912189,0.22457759],[1,0,-1,1],[9E+09,9E+09,9E+09,9E+09,9E+09,9E+09]];
	CONST robtarget Target_debavurare33:=[[70.188915319,1029.778488373,2213.889],[0.970550763,-0.019647992,0.084912189,0.22457759],[0,0,-1,1],[9E+09,9E+09,9E+09,9E+09,9E+09,9E+09]];
	CONST robtarget Target_debavurare34:=[[76.541263714,1032.884558215,2210.960067812],[0.970550763,-0.019647992,0.084912189,0.22457759],[0,0,-1,1],[9E+09,9E+09,9E+09,9E+09,9E+09,9E+09]];
	CONST robtarget Target_debavurare35:=[[79.172492573,1034.171134469,2203.889],[0.626241041,-0.172693565,0.74632501,0.144907108],[1,1,-2,1],[9E+09,9E+09,9E+09,9E+09,9E+09,9E+09]];
	CONST robtarget Target_debavurare36:=[[79.172492573,1034.171134469,672.279996312],[0.626241041,-0.172693565,0.74632501,0.144907108],[1,0,-1,1],[9E+09,9E+09,9E+09,9E+09,9E+09,9E+09]];
	CONST robtarget Target_debavurare37:=[[77.070734753,1033.143450506,665.852120215],[0.626241041,-0.172693565,0.74632501,0.144907108],[1,0,-1,1],[9E+09,9E+09,9E+09,9E+09,9E+09,9E+09]];
	CONST robtarget Target_debavurare38:=[[71.748897138,1030.541263363,662.431918782],[0.626241041,-0.172693565,0.74632501,0.144907108],[1,0,-1,1],[9E+09,9E+09,9E+09,9E+09,9E+09,9E+09]];
	CONST robtarget Target_debavurare39:=[[-91.515475248,950.710858642,630.386873665],[0.626241041,-0.172693565,0.74632501,0.144907108],[1,1,-1,1],[9E+09,9E+09,9E+09,9E+09,9E+09,9E+09]];
	CONST robtarget Target_debavurare40:=[[-82.17325952,955.27886605,571.409990938],[0.626241041,-0.172693565,0.74632501,0.144907108],[1,1,-1,1],[9E+09,9E+09,9E+09,9E+09,9E+09,9E+09]];
	CONST robtarget Target_debavurare41:=[[235.647161917,962.336296138,604.766182313],[0.626241041,-0.172693565,0.74632501,0.144907108],[0,0,-1,1],[9E+09,9E+09,9E+09,9E+09,9E+09,9E+09]];
	CONST robtarget Target_debavurare42:=[[222.398190082,1104.203348059,561.899220237],[0.320706496,-0.564932078,0.425266677,0.630196274],[0,1,-2,0],[9E+09,9E+09,9E+09,9E+09,9E+09,9E+09]];
	CONST robtarget Target_debavurare43:=[[4.592265391,1019.966932715,523.466438018],[0.425266678,-0.630196274,0.320706495,0.564932078],[0,1,-2,0],[9E+09,9E+09,9E+09,9E+09,9E+09,9E+09]];
	CONST robtarget Target_debavurare44:=[[-67.51635848,984.708409724,538.596152517],[0.425266678,-0.630196274,0.320706495,0.564932078],[0,1,-2,0],[9E+09,9E+09,9E+09,9E+09,9E+09,9E+09]];
	CONST robtarget Target_debavurare45:=[[-74.04786326,1009.140395264,511.008322261],[0.425266678,-0.630196274,0.320706495,0.564932078],[0,1,-2,0],[9E+09,9E+09,9E+09,9E+09,9E+09,9E+09]];
	CONST robtarget Target_debavurare46:=[[-57.20170243,983.09209564,490.071182954],[0.425266678,-0.630196274,0.320706495,0.564932078],[0,1,-2,0],[9E+09,9E+09,9E+09,9E+09,9E+09,9E+09]];
	CONST robtarget Target_debavurare47:=[[-53.184944606,964.090299134,516.943595123],[0.425266678,-0.630196274,0.320706495,0.564932078],[0,1,-2,0],[9E+09,9E+09,9E+09,9E+09,9E+09,9E+09]];
	CONST robtarget Target_debavurare48:=[[-67.51635848,984.708409724,538.596152517],[0.425266678,-0.630196274,0.320706495,0.564932078],[0,1,-2,0],[9E+09,9E+09,9E+09,9E+09,9E+09,9E+09]];
	CONST robtarget Target_debavurare49:=[[380.563228786,1203.803208398,695.774665043],[0.425266678,-0.630196274,0.320706495,0.564932078],[0,1,-2,0],[9E+09,9E+09,9E+09,9E+09,9E+09,9E+09]];
	CONST robtarget Target_debavurare50:=[[236.855316057,878.977367128,797.279996312],[0.626241041,-0.172693565,0.74632501,0.144907108],[0,0,-1,1],[9E+09,9E+09,9E+09,9E+09,9E+09,9E+09]];
	CONST robtarget Target_debavurare51:=[[-106.574951523,844.917671275,913.754533399],[0.626241041,-0.172693565,0.74632501,0.144907108],[1,1,-1,1],[9E+09,9E+09,9E+09,9E+09,9E+09,9E+09]];
	CONST robtarget Target_debavurare52:=[[-251.957733199,755.881530829,797.279996312],[0.626241041,-0.172693565,0.74632501,0.144907108],[1,1,-1,1],[9E+09,9E+09,9E+09,9E+09,9E+09,9E+09]];
	CONST robtarget Target_debavurare53:=[[-306.602704629,845.540941159,797.279996312],[0.626241041,-0.172693565,0.74632501,0.144907108],[1,1,-1,1],[9E+09,9E+09,9E+09,9E+09,9E+09,9E+09]];
	CONST robtarget Target_debavurare54:=[[-55.581166233,968.281443027,797.279996312],[0.626241041,-0.172693565,0.74632501,0.144907108],[1,1,-1,1],[9E+09,9E+09,9E+09,9E+09,9E+09,9E+09]];
	CONST robtarget Target_debavurare55:=[[-55.581166233,968.281443027,1260.498003688],[0.626241041,-0.172693565,0.74632501,0.144907108],[1,1,-1,1],[9E+09,9E+09,9E+09,9E+09,9E+09,9E+09]];
	CONST robtarget Target_debavurare56:=[[-57.682924053,967.253759063,1266.925879785],[0.626241041,-0.172693565,0.74632501,0.144907108],[1,1,-1,1],[9E+09,9E+09,9E+09,9E+09,9E+09,9E+09]];
	CONST robtarget Target_debavurare57:=[[-63.004761668,964.65157192,1270.346081218],[0.626241041,-0.172693565,0.74632501,0.144907108],[1,1,-1,1],[9E+09,9E+09,9E+09,9E+09,9E+09,9E+09]];
	CONST robtarget Target_debavurare58:=[[-326.648465665,835.739285151,1321.480905624],[0.626241041,-0.172693565,0.74632501,0.144907108],[1,1,-1,1],[9E+09,9E+09,9E+09,9E+09,9E+09,9E+09]];
	CONST robtarget Target_debavurare59:=[[-587.172206023,708.352548362,1270.346081218],[0.626241041,-0.172693565,0.74632501,0.144907108],[1,1,-1,1],[9E+09,9E+09,9E+09,9E+09,9E+09,9E+09]];
	CONST robtarget Target_debavurare60:=[[-592.494043638,705.75036122,1266.925879785],[0.626241041,-0.172693565,0.74632501,0.144907108],[1,1,-1,1],[9E+09,9E+09,9E+09,9E+09,9E+09,9E+09]];
	CONST robtarget Target_debavurare61:=[[-594.595801457,704.722677256,1260.498003688],[0.626241041,-0.172693565,0.74632501,0.144907108],[1,1,-1,1],[9E+09,9E+09,9E+09,9E+09,9E+09,9E+09]];
	CONST robtarget Target_debavurare62:=[[-594.595801457,704.722677256,797.279996312],[0.626241041,-0.172693565,0.74632501,0.144907108],[1,1,-1,1],[9E+09,9E+09,9E+09,9E+09,9E+09,9E+09]];
	CONST robtarget Target_debavurare63:=[[-592.494043638,705.75036122,790.852120215],[0.626241041,-0.172693565,0.74632501,0.144907108],[1,1,-1,1],[9E+09,9E+09,9E+09,9E+09,9E+09,9E+09]];
	CONST robtarget Target_debavurare64:=[[-587.172206023,708.352548362,787.431918782],[0.626241041,-0.172693565,0.74632501,0.144907108],[1,1,-1,1],[9E+09,9E+09,9E+09,9E+09,9E+09,9E+09]];
	CONST robtarget Target_debavurare65:=[[-323.528502026,837.264835131,736.297094376],[0.626241041,-0.172693565,0.74632501,0.144907108],[1,1,-1,1],[9E+09,9E+09,9E+09,9E+09,9E+09,9E+09]];
	CONST robtarget Target_debavurare66:=[[-63.004761668,964.65157192,787.431918782],[0.626241041,-0.172693565,0.74632501,0.144907108],[1,1,-1,1],[9E+09,9E+09,9E+09,9E+09,9E+09,9E+09]];
	CONST robtarget Target_debavurare67:=[[-57.682924053,967.253759063,790.852120215],[0.626241041,-0.172693565,0.74632501,0.144907108],[1,1,-1,1],[9E+09,9E+09,9E+09,9E+09,9E+09,9E+09]];
	CONST robtarget Target_debavurare68:=[[-55.581166233,968.281443027,797.279996312],[0.626241041,-0.172693565,0.74632501,0.144907108],[1,1,-1,1],[9E+09,9E+09,9E+09,9E+09,9E+09,9E+09]];
	CONST robtarget Target_debavurare69:=[[-4.129380996,863.055327059,797.279996312],[0.626241041,-0.172693565,0.74632501,0.144907108],[1,1,-1,1],[9E+09,9E+09,9E+09,9E+09,9E+09,9E+09]];
	CONST robtarget Target_evacuare12:=[[353.286050265,-1090.926157105,1000],[0,0,1,-0.000000001],[-1,0,-1,0],[9E+09,9E+09,9E+09,9E+09,9E+09,9E+09]];
	CONST robtarget Target_control1:=[[1164.241304795,1065.453076327,1110.91287582],[0,0.848311443,-0.529497588,0],[0,0,-1,0],[9E+09,9E+09,9E+09,9E+09,9E+09,9E+09]];
	CONST robtarget Target_control2:=[[561.343174474,770.657579762,1105.422922565],[0,0.848311443,-0.529497588,0],[0,0,-1,0],[9E+09,9E+09,9E+09,9E+09,9E+09,9E+09]];
	CONST robtarget Target_control3:=[[-352.181570531,474.725664361,1108.429867517],[0.630196274,-0.425266678,-0.564932078,-0.320706495],[1,-2,-1,0],[9E+09,9E+09,9E+09,9E+09,9E+09,9E+09]];
	CONST robtarget Target_control4:=[[-965.595492909,398.655755176,510.210088752],[0.630196274,-0.425266678,-0.564932078,-0.320706495],[1,-2,-1,0],[9E+09,9E+09,9E+09,9E+09,9E+09,9E+09]];
	CONST robtarget Target_control5:=[[-676.765426106,531.291262028,504.173173014],[0.630196274,-0.425266678,-0.564932078,-0.320706495],[1,-2,-1,0],[9E+09,9E+09,9E+09,9E+09,9E+09,9E+09]];
	CONST robtarget Target_control6:=[[-676.765426106,531.291262028,2203.889],[0.630196274,-0.425266678,-0.564932078,-0.320706495],[1,-1,-2,0],[9E+09,9E+09,9E+09,9E+09,9E+09,9E+09]];
	CONST robtarget Target_control7:=[[-542.0117673,597.180953471,2203.889],[0.630196274,-0.425266678,-0.564932078,-0.320706495],[1,-1,-2,0],[9E+09,9E+09,9E+09,9E+09,9E+09,9E+09]];
	CONST robtarget Target_control8:=[[-534.588171866,600.810824577,1457.431918782],[0.630196274,-0.425266678,-0.564932078,-0.320706495],[1,-1,-1,0],[9E+09,9E+09,9E+09,9E+09,9E+09,9E+09]];
	CONST robtarget Target_control9:=[[-270.944467869,729.723111346,1406.297094376],[0.630196274,-0.425266678,-0.564932078,-0.320706495],[1,-1,-1,1],[9E+09,9E+09,9E+09,9E+09,9E+09,9E+09]];
	CONST robtarget Target_control10:=[[-10.420727511,857.109848135,1457.431918782],[0.630196274,-0.425266678,-0.564932078,-0.320706495],[0,-1,-1,1],[9E+09,9E+09,9E+09,9E+09,9E+09,9E+09]];
	CONST robtarget Target_control11:=[[-2.997132076,860.739719242,2203.889],[0.630196274,-0.425266678,-0.564932078,-0.320706495],[0,-2,-1,1],[9E+09,9E+09,9E+09,9E+09,9E+09,9E+09]];
	CONST robtarget Target_control12:=[[131.75652673,926.629410684,2203.889],[0.630196274,-0.425266678,-0.564932078,-0.320706495],[0,-2,-1,1],[9E+09,9E+09,9E+09,9E+09,9E+09,9E+09]];
	CONST robtarget Target_control13:=[[131.75652673,926.629410684,672.279996312],[0.630196274,-0.425266678,-0.564932078,-0.320706495],[0,-1,-2,1],[9E+09,9E+09,9E+09,9E+09,9E+09,9E+09]];
	CONST robtarget Target_control14:=[[-38.931441091,843.169134857,630.386873665],[0.630196274,-0.425266678,-0.564932078,-0.320706495],[0,-1,-2,1],[9E+09,9E+09,9E+09,9E+09,9E+09,9E+09]];
	CONST robtarget Target_control15:=[[-29.589225363,847.737142265,571.409990938],[0.630196274,-0.425266678,-0.564932078,-0.320706495],[0,-1,-2,1],[9E+09,9E+09,9E+09,9E+09,9E+09,9E+09]];
	CONST robtarget Target_control16:=[[-53.990917366,737.37594749,913.754533399],[0.630196274,-0.425266678,-0.564932078,-0.320706495],[0,-1,-2,1],[9E+09,9E+09,9E+09,9E+09,9E+09,9E+09]];
	CONST robtarget Target_control17:=[[-2.997132076,860.739719242,797.279996312],[0.630196274,-0.425266678,-0.564932078,-0.320706495],[0,-1,-2,1],[9E+09,9E+09,9E+09,9E+09,9E+09,9E+09]];
	CONST robtarget Target_control18:=[[-2.997132076,860.739719242,1260.498003688],[0.630196274,-0.425266678,-0.564932078,-0.320706495],[0,-1,-2,1],[9E+09,9E+09,9E+09,9E+09,9E+09,9E+09]];
	CONST robtarget Target_control19:=[[-274.064431508,728.197561366,1321.480905624],[0.630196274,-0.425266678,-0.564932078,-0.320706495],[1,-1,-2,1],[9E+09,9E+09,9E+09,9E+09,9E+09,9E+09]];
	CONST robtarget Target_control20:=[[-542.0117673,597.180953471,1260.498003688],[0.630196274,-0.425266678,-0.564932078,-0.320706495],[1,-2,-1,0],[9E+09,9E+09,9E+09,9E+09,9E+09,9E+09]];
	CONST robtarget Target_control21:=[[-542.0117673,597.180953471,797.279996312],[0.630196274,-0.425266678,-0.564932078,-0.320706495],[1,-2,-1,0],[9E+09,9E+09,9E+09,9E+09,9E+09,9E+09]];
	CONST robtarget Target_control22:=[[-270.944467869,729.723111346,736.297094376],[0.630196274,-0.425266678,-0.564932078,-0.320706495],[1,-1,-2,1],[9E+09,9E+09,9E+09,9E+09,9E+09,9E+09]];
	CONST robtarget Target_control23:=[[-10.420727511,857.109848135,787.431918782],[0.630196274,-0.425266678,-0.564932078,-0.320706495],[0,-1,-2,1],[9E+09,9E+09,9E+09,9E+09,9E+09,9E+09]];
	CONST robtarget Target_control24:=[[-2.997132076,860.739719242,797.279996312],[0.630196274,-0.425266678,-0.564932078,-0.320706495],[0,-1,-2,1],[9E+09,9E+09,9E+09,9E+09,9E+09,9E+09]];
	CONST robtarget Target_control25:=[[48.454653161,755.513603274,797.279996312],[0.630196274,-0.425266678,-0.564932078,-0.320706495],[0,-1,-2,1],[9E+09,9E+09,9E+09,9E+09,9E+09,9E+09]];
	CONST robtarget Target_control26:=[[389.997020927,869.040623857,1101.572770211],[0.630196274,-0.425266678,-0.564932078,-0.320706495],[0,-1,-2,1],[9E+09,9E+09,9E+09,9E+09,9E+09,9E+09]];
	CONST robtarget Target_evacuare1:=[[-297.408117168,261.539979913,1840.929204997],[0.159406928,0.159406928,-0.688904515,-0.688904516],[0,0,0,4],[9E+09,9E+09,9E+09,9E+09,9E+09,9E+09]];
	CONST robtarget Target_evacuare2:=[[-117.985307131,412.947477324,1336.176966578],[0.159406928,0.159406928,-0.688904515,-0.688904516],[0,0,0,0],[9E+09,9E+09,9E+09,9E+09,9E+09,9E+09]];
	CONST robtarget Target_evacuare3:=[[-320.695795916,827.518853271,1336.176966578],[0.159406928,0.159406928,-0.688904515,-0.688904516],[1,0,0,0],[9E+09,9E+09,9E+09,9E+09,9E+09,9E+09]];
	CONST robtarget Target_evacuare4:=[[-117.985307131,412.947477324,1336.176966578],[0.159406928,0.159406928,-0.688904515,-0.688904516],[0,0,0,0],[9E+09,9E+09,9E+09,9E+09,9E+09,9E+09]];
	CONST robtarget Target_evacuare5:=[[1072.781898944,-59.825918958,1479.636846222],[0.374411334,0.374411335,0.599846774,0.599846775],[-1,1,-1,0],[9E+09,9E+09,9E+09,9E+09,9E+09,9E+09]];
	CONST robtarget Target_evacuare6:=[[1215.425844801,-519.48484737,1533.087792477],[0.374411334,0.374411335,0.599846774,0.599846775],[-1,1,-1,0],[9E+09,9E+09,9E+09,9E+09,9E+09,9E+09]];
	CONST robtarget Target_evacuare7:=[[71.368530681,-1273.53877769,1533.087792477],[0.688904515,0.688904516,0.159406928,0.159406928],[-2,1,-1,0],[9E+09,9E+09,9E+09,9E+09,9E+09,9E+09]];
	CONST robtarget Target_evacuare8:=[[-427.431513587,-1517.434055188,1533.087792477],[0.000000001,0.974258109,0.225435439,0],[-2,-1,0,0],[9E+09,9E+09,9E+09,9E+09,9E+09,9E+09]];
	CONST robtarget Target_evacuare9:=[[-935.838539063,-1766.02680089,1533.087792477],[-0.000000001,0.974258109,0.225435439,0],[-2,0,0,0],[9E+09,9E+09,9E+09,9E+09,9E+09,9E+09]];
	CONST robtarget Target_evacuare10:=[[-994.92710219,-1794.918982569,917.887564527],[0.000000001,0.974258109,0.225435439,0],[-2,-1,0,0],[9E+09,9E+09,9E+09,9E+09,9E+09,9E+09]];
	CONST robtarget Target_evacuare11:=[[-994.92710219,-1794.918982569,697.821327506],[-0.000000001,0.974258109,0.225435439,0],[-2,0,0,0],[9E+09,9E+09,9E+09,9E+09,9E+09,9E+09]];
	CONST robtarget Target_decuplare_ATI1:=[[389.997020927,869.040623857,1101.572770211],[0.630196274,-0.425266678,-0.564932078,-0.320706495],[0,1,0,0],[9E+09,9E+09,9E+09,9E+09,9E+09,9E+09]];
	CONST robtarget Target_decuplare_ATI2:=[[504.928038476,563.849286682,1069.091100494],[0,0.848311443,-0.529497588,0],[0,0,-1,0],[9E+09,9E+09,9E+09,9E+09,9E+09,9E+09]];
	CONST robtarget Target_decuplare_ATI3:=[[561.343174474,770.657579762,1105.422922565],[0,0.848311443,-0.529497588,0],[0,0,-1,0],[9E+09,9E+09,9E+09,9E+09,9E+09,9E+09]];
	CONST robtarget Target_decuplare_ATI4:=[[1164.241304795,1065.453076327,1110.91287582],[0,0.848311443,-0.529497588,0],[0,0,-1,0],[9E+09,9E+09,9E+09,9E+09,9E+09,9E+09]];
	CONST robtarget Target_decuplare_ATI5:=[[1164.456250233,1065.58489233,1000],[0,0.848311443,-0.529497588,0],[0,0,-1,0],[9E+09,9E+09,9E+09,9E+09,9E+09,9E+09]];
	CONST robtarget Target_schimbare_efectori1:=[[-176.063589295,-890.179717053,2221.711117045],[0.579227966,0.405579787,-0.5,-0.5],[1,0,0,4],[9E+09,9E+09,9E+09,9E+09,9E+09,9E+09]];
	CONST robtarget Target_schimbare_efectori2:=[[-549.798887424,-878.736368632,2286.609570489],[0.69636424,-0.122787804,0,-0.707106781],[1,-1,0,1],[9E+09,9E+09,9E+09,9E+09,9E+09,9E+09]];
	CONST robtarget Target_schimbare_efectori3:=[[-658.456780387,304.505009965,2066.113793534],[0.69636424,-0.122787804,0,-0.707106781],[0,-1,1,1],[9E+09,9E+09,9E+09,9E+09,9E+09,9E+09]];
	CONST robtarget Target_schimbare_efectori4:=[[-690.279328221,273.165917946,1888.380971862],[0.69636424,-0.122787804,0,-0.707106781],[0,-1,1,1],[9E+09,9E+09,9E+09,9E+09,9E+09,9E+09]];
	CONST robtarget Target_schimbare_efectori5:=[[779.908229606,894.538776646,1570.162539077],[0.225435439,0,0,-0.974258109],[0,0,1,1],[9E+09,9E+09,9E+09,9E+09,9E+09,9E+09]];
	CONST robtarget Target_schimbare_efectori6:=[[367.891360431,693.077349856,1324.929850073],[0,0.848311443,-0.529497588,0],[0,0,-1,0],[9E+09,9E+09,9E+09,9E+09,9E+09,9E+09]];
	CONST robtarget Target_schimbare_efectori7:=[[553.518951213,783.842563864,1017.503826288],[0,0.848311443,-0.529497588,0],[0,0,-1,0],[9E+09,9E+09,9E+09,9E+09,9E+09,9E+09]];
	CONST robtarget Target_schimbare_efectori8:=[[1164.456250233,1065.58489233,1033.237043133],[0,0.848311443,-0.529497588,0],[0,0,-1,0],[9E+09,9E+09,9E+09,9E+09,9E+09,9E+09]];
	CONST robtarget Target_schimbare_efectori9:=[[1164.456250233,1065.58489233,1000],[0,0.848311443,-0.529497588,0],[0,0,-1,0],[9E+09,9E+09,9E+09,9E+09,9E+09,9E+09]];
	CONST robtarget Target_schimbare_efectori11:=[[561.343174474,770.657579762,1105.422922565],[0,0.848311443,-0.529497588,0],[0,0,-1,0],[9E+09,9E+09,9E+09,9E+09,9E+09,9E+09]];
	CONST robtarget Target_cuplare_V1:=[[779.908229606,894.538776646,1570.162539077],[0.225435439,0,0,-0.974258109],[0,0,1,1],[9E+09,9E+09,9E+09,9E+09,9E+09,9E+09]];
	CONST robtarget Target_cuplare_V2:=[[766.154301146,968.592405176,2185.609751442],[0.225435439,0,0,-0.974258109],[0,0,1,1],[9E+09,9E+09,9E+09,9E+09,9E+09,9E+09]];
	CONST robtarget Target_cuplare_V3:=[[766.154301146,968.592405176,2185.609751442],[0.225435439,0,0,-0.974258109],[0,0,1,1],[9E+09,9E+09,9E+09,9E+09,9E+09,9E+09]];
	CONST robtarget Target_cuplare_V4:=[[766.154301147,968.592405175,2579.975738982],[0.225435439,0,0,-0.974258109],[0,0,1,1],[9E+09,9E+09,9E+09,9E+09,9E+09,9E+09]];
	CONST robtarget Target_cuplare_V5:=[[-148.366452112,98.986292765,2610.344805667],[0.159406928,0.159406928,-0.688904515,-0.688904516],[1,0,0,4],[9E+09,9E+09,9E+09,9E+09,9E+09,9E+09]];
    PROC Home()
        SetDO\SDelay:=0.1,do_cupleaza_ATI,0;
	    SetDO\SDelay:=0.1,do_cupleaza_V,1;
	    MoveJ Target_evacuare12,v500,z100,Flansa_Cuplare\WObj:=wobj_alimentare;
        TPWrite "Se asteapta aducerea piesei pe masa în pozitie centrata";
	    WaitDI DI_S2_piesa_pe_masa,1;
	    Path1_Preluare_piesa;
	ENDPROC
	PROC Path1_Preluare_piesa()
        TPWrite "Efectuare proces de preluare a piesei de pe masa";
	    MoveJ Target_preluare_piesa1,v1000,z100,Tooldata_TCP_VAC\WObj:=wobj_alimentare;
	    MoveJ Target_preluare_piesa2,v600,z100,Tooldata_TCP_VAC\WObj:=wobj_alimentare;
	    WaitTime\InPos,0.5;
	    SetDO\SDelay:=0,DO_piesa_gata,0;
	    SetDO\SDelay:=1,DO_S7_piesa_efector_V,1;
        TPWrite "Piesa este preluata de efectotul vacuumatic";
	    WaitTime\InPos,1;
	    MoveJ Target_preluare_piesa3,v600,z100,Tooldata_TCP_VAC\WObj:=wobj_alimentare;
	    MoveJ Target_preluare_piesa4,v600,z100,Tooldata_TCP_VAC\WObj:=wobj_alimentare;
	    MoveJ Target_preluare_piesa5,v600,z100,Tooldata_TCP_VAC\WObj:=wobj_alimentare;
	    MoveJ Target_preluare_piesa6,v600,z100,Tooldata_TCP_VAC\WObj:=wobj_alimentare;
	    MoveJ Target_preluare_piesa7,v600,z100,Tooldata_TCP_VAC\WObj:=wobj_alimentare;
	    MoveJ Target_preluare_piesa8,v1000,z100,Tooldata_TCP_VAC\WObj:=wobj_alimentare;
	    WaitTime\InPos,0.5;
	    SetDO\SDelay:=0.5,DO_S7_piesa_efector_V,0;
	    SetDO\SDelay:=0.5,DO_S4_Sistem_fixare,1;
        TPWrite "Piesa este fixata în suportul de fixare";
	    WaitTime\InPos,1;
	    MoveJ Target_preluare_piesa7,v1000,z100,Tooldata_TCP_VAC\WObj:=wobj_alimentare;
	    MoveJ Target_preluare_piesa9,v1000,z100,Tooldata_TCP_VAC\WObj:=wobj_alimentare;
	    Path2_Schimbare_efectori;
	ENDPROC
    PROC Path2_Schimbare_efectori()
        TPWrite "Efectuare proces de schimbare a efectorilor";
	    MoveJ Target_schimbare_efectori1,v800,z100,Tooldata_TCP_VAC\WObj:=wobj_alimentare;
	    MoveJ Target_schimbare_efectori2,v800,z100,Tooldata_TCP_VAC\WObj:=wobj_alimentare;
	    MoveL Target_schimbare_efectori3,v600,z100,Tooldata_TCP_VAC\WObj:=wobj_alimentare;
	    MoveJ Target_schimbare_efectori4,v400,z100,Tooldata_TCP_VAC\WObj:=wobj_alimentare;
	    WaitTime\InPos,0.5;
	    SetDO\SDelay:=1,do_cupleaza_V,0;
        TPWrite "Efector vacuumatic decuplat";
	    WaitTime\InPos,1;
	    SetDO\SDelay:=0,DO_deschide_cutie,1;
        TPWrite "Sistem de protectie ATI deschis";
	    MoveJ Target_schimbare_efectori5,v800,z100,Flansa_Cuplare\WObj:=wobj_schimbare_efectori;
	    MoveJ Target_schimbare_efectori6,v800,z100,Flansa_Cuplare\WObj:=wobj_schimbare_efectori;
	    MoveJ Target_schimbare_efectori7,v800,z100,Flansa_Cuplare\WObj:=wobj_schimbare_efectori;
	    MoveJ Target_schimbare_efectori8,v500,z100,Flansa_Cuplare\WObj:=wobj_schimbare_efectori;
	    MoveJ Target_schimbare_efectori9,v300,z50,Flansa_Cuplare\WObj:=wobj_schimbare_efectori;
	    WaitTime\InPos,0.5;
	    SetDO\SDelay:=1,do_cupleaza_ATI,1;
        TPWrite "Efector ATI cuplat";
	    WaitTime\InPos,1;
	    MoveJ Target_decuplare_ATI4,v300,z100,Flansa_Cuplare\WObj:=wobj_schimbare_efectori;
	    MoveJ Target_schimbare_efectori11,v800,z100,Flansa_Cuplare\WObj:=wobj_schimbare_efectori;
	    Path3_Debavurare;
	ENDPROC
	PROC Path3_Debavurare()
        TPWrite "Efectuare proces de debvurare a reperului";
	    MoveJ Target_debavurare1,v500,z100,Flansa_Cuplare\WObj:=wobj_schimbare_efectori;
	    SetDO\SDelay:=0,DO_deschide_cutie,0;
        TPWrite "Sistem de protectie ATI închis";
	    MoveJ Target_debavurare2,v500,z100,Flansa_Cuplare\WObj:=wobj_schimbare_efectori;
	    MoveJ Target_debavurare3,v500,z100,Flansa_Cuplare\WObj:=wobj_schimbare_efectori;
	    MoveJ Target_debavurare4,v1000,z100,Tooldata_TCP_ATI\WObj:=wobj_schimbare_efectori;
	    MoveJ Target_debavurare5,v1000,z100,Tooldata_TCP_ATI\WObj:=wobj_schimbare_efectori;
	    MoveC Target_debavurare6,Target_debavurare7,v1000,z100,Tooldata_TCP_ATI\WObj:=wobj_schimbare_efectori;
	    MoveC Target_debavurare8,Target_debavurare9,v1000,z100,Tooldata_TCP_ATI\WObj:=wobj_schimbare_efectori;
	    MoveJ Target_debavurare10,v1000,z100,Tooldata_TCP_ATI\WObj:=wobj_schimbare_efectori;
	    MoveJ Target_debavurare11,v1000,z100,Tooldata_TCP_ATI\WObj:=wobj_schimbare_efectori;
	    MoveJ Target_debavurare12,v1000,z100,Tooldata_TCP_ATI\WObj:=wobj_schimbare_efectori;
	    MoveL Target_debavurare13,v1000,z100,Tooldata_TCP_ATI\WObj:=wobj_schimbare_efectori;
	    MoveL Target_debavurare14,v1000,z100,Tooldata_TCP_ATI\WObj:=wobj_schimbare_efectori;
	    MoveL Target_debavurare15,v1000,z100,Tooldata_TCP_ATI\WObj:=wobj_schimbare_efectori;
	    MoveL Target_debavurare16,v1000,z100,Tooldata_TCP_ATI\WObj:=wobj_schimbare_efectori;
	    MoveL Target_debavurare17,v1000,z100,Tooldata_TCP_ATI\WObj:=wobj_schimbare_efectori;
	    MoveL Target_debavurare18,v1000,z100,Tooldata_TCP_ATI\WObj:=wobj_schimbare_efectori;
	    MoveL Target_debavurare19,v1000,z100,Tooldata_TCP_ATI\WObj:=wobj_schimbare_efectori;
	    MoveL Target_debavurare20,v1000,z100,Tooldata_TCP_ATI\WObj:=wobj_schimbare_efectori;
	    MoveL Target_debavurare21,v1000,z100,Tooldata_TCP_ATI\WObj:=wobj_schimbare_efectori;
	    MoveL Target_debavurare22,v1000,z100,Tooldata_TCP_ATI\WObj:=wobj_schimbare_efectori;
	    MoveL Target_debavurare23,v1000,z100,Tooldata_TCP_ATI\WObj:=wobj_schimbare_efectori;
	    MoveL Target_debavurare24,v1000,z100,Tooldata_TCP_ATI\WObj:=wobj_schimbare_efectori;
	    MoveL Target_debavurare25,v1000,z100,Tooldata_TCP_ATI\WObj:=wobj_schimbare_efectori;
	    MoveL Target_debavurare26,v1000,z100,Tooldata_TCP_ATI\WObj:=wobj_schimbare_efectori;
	    MoveL Target_debavurare27,v1000,z100,Tooldata_TCP_ATI\WObj:=wobj_schimbare_efectori;
	    MoveL Target_debavurare28,v1000,z100,Tooldata_TCP_ATI\WObj:=wobj_schimbare_efectori;
	    MoveL Target_debavurare29,v1000,z100,Tooldata_TCP_ATI\WObj:=wobj_schimbare_efectori;
	    MoveL Target_debavurare30,v1000,z100,Tooldata_TCP_ATI\WObj:=wobj_schimbare_efectori;
	    MoveL Target_debavurare31,v1000,z100,Tooldata_TCP_ATI\WObj:=wobj_schimbare_efectori;
	    MoveL Target_debavurare32,v1000,z100,Tooldata_TCP_ATI\WObj:=wobj_schimbare_efectori;
	    MoveL Target_debavurare33,v1000,z100,Tooldata_TCP_ATI\WObj:=wobj_schimbare_efectori;
	    MoveJ Target_debavurare34,v1000,z100,Tooldata_TCP_ATI\WObj:=wobj_schimbare_efectori;
	    MoveJ Target_debavurare35,v1000,z100,Tooldata_TCP_ATI\WObj:=wobj_schimbare_efectori;
	    MoveL Target_debavurare36,v1000,z100,Tooldata_TCP_ATI\WObj:=wobj_schimbare_efectori;
	    MoveL Target_debavurare37,v1000,z100,Tooldata_TCP_ATI\WObj:=wobj_schimbare_efectori;
	    MoveL Target_debavurare38,v1000,z100,Tooldata_TCP_ATI\WObj:=wobj_schimbare_efectori;
	    MoveL Target_debavurare39,v1000,z100,Tooldata_TCP_ATI\WObj:=wobj_schimbare_efectori;
	    MoveL Target_debavurare40,v1000,z100,Tooldata_TCP_ATI\WObj:=wobj_schimbare_efectori;
	    MoveJ Target_debavurare41,v1000,z100,Tooldata_TCP_ATI\WObj:=wobj_schimbare_efectori;
	    MoveJ Target_debavurare42,v1000,z100,Tooldata_TCP_ATI\WObj:=wobj_schimbare_efectori;
	    MoveJ Target_debavurare43,v1000,z100,Tooldata_TCP_ATI\WObj:=wobj_schimbare_efectori;
	    MoveJ Target_debavurare44,v1000,z100,Tooldata_TCP_ATI\WObj:=wobj_schimbare_efectori;
	    MoveC Target_debavurare45,Target_debavurare46,v1000,z100,Tooldata_TCP_ATI\WObj:=wobj_schimbare_efectori;
	    MoveC Target_debavurare47,Target_debavurare48,v1000,z100,Tooldata_TCP_ATI\WObj:=wobj_schimbare_efectori;
	    MoveJ Target_debavurare49,v1000,z100,Tooldata_TCP_ATI\WObj:=wobj_schimbare_efectori;
	    MoveJ Target_debavurare50,v1000,z100,Tooldata_TCP_ATI\WObj:=wobj_schimbare_efectori;
	    MoveJ Target_debavurare51,v1000,z100,Tooldata_TCP_ATI\WObj:=wobj_schimbare_efectori;
	    MoveJ Target_debavurare52,v1000,z100,Tooldata_TCP_ATI\WObj:=wobj_schimbare_efectori;
	    MoveJ Target_debavurare53,v1000,z100,Tooldata_TCP_ATI\WObj:=wobj_schimbare_efectori;
	    MoveJ Target_debavurare54,v1000,z100,Tooldata_TCP_ATI\WObj:=wobj_schimbare_efectori;
	    MoveL Target_debavurare55,v1000,z100,Tooldata_TCP_ATI\WObj:=wobj_schimbare_efectori;
	    MoveL Target_debavurare56,v1000,z100,Tooldata_TCP_ATI\WObj:=wobj_schimbare_efectori;
	    MoveL Target_debavurare57,v1000,z100,Tooldata_TCP_ATI\WObj:=wobj_schimbare_efectori;
	    MoveL Target_debavurare58,v1000,z100,Tooldata_TCP_ATI\WObj:=wobj_schimbare_efectori;
	    MoveL Target_debavurare59,v1000,z100,Tooldata_TCP_ATI\WObj:=wobj_schimbare_efectori;
	    MoveL Target_debavurare60,v1000,z100,Tooldata_TCP_ATI\WObj:=wobj_schimbare_efectori;
	    MoveL Target_debavurare61,v1000,z100,Tooldata_TCP_ATI\WObj:=wobj_schimbare_efectori;
	    MoveL Target_debavurare62,v1000,z100,Tooldata_TCP_ATI\WObj:=wobj_schimbare_efectori;
	    MoveL Target_debavurare63,v1000,z100,Tooldata_TCP_ATI\WObj:=wobj_schimbare_efectori;
	    MoveL Target_debavurare64,v1000,z100,Tooldata_TCP_ATI\WObj:=wobj_schimbare_efectori;
	    MoveL Target_debavurare65,v1000,z100,Tooldata_TCP_ATI\WObj:=wobj_schimbare_efectori;
	    MoveL Target_debavurare66,v1000,z100,Tooldata_TCP_ATI\WObj:=wobj_schimbare_efectori;
	    MoveL Target_debavurare67,v1000,z100,Tooldata_TCP_ATI\WObj:=wobj_schimbare_efectori;
	    MoveL Target_debavurare68,v1000,z100,Tooldata_TCP_ATI\WObj:=wobj_schimbare_efectori;
	    MoveJ Target_debavurare69,v1000,z100,Tooldata_TCP_ATI\WObj:=wobj_schimbare_efectori;
	    Path4_Decuplare_ATI;
	ENDPROC
	PROC Path4_Decuplare_ATI()
	    SetDO\SDelay:=0,DO_deschide_cutie,1;
        TPWrite "Sistem de protectie ATI deschis";
	    MoveJ Target_decuplare_ATI1,v500,z100,Flansa_Cuplare\WObj:=wobj_schimbare_efectori;
	    MoveJ Target_decuplare_ATI2,v500,z100,Flansa_Cuplare\WObj:=wobj_schimbare_efectori;
	    MoveJ Target_decuplare_ATI3,v500,z100,Flansa_Cuplare\WObj:=wobj_schimbare_efectori;
	    MoveJ Target_decuplare_ATI4,v500,z100,Flansa_Cuplare\WObj:=wobj_schimbare_efectori;
	    MoveJ Target_decuplare_ATI5,v500,z100,Flansa_Cuplare\WObj:=wobj_control;
	    WaitTime\InPos,0.5;
	    SetDO\SDelay:=1,do_cupleaza_ATI,0;
        TPWrite "Efector ATI decuplat";
        WaitTime\InPos,1;
	    Path5_Control_vizual;
	ENDPROC
	PROC Path5_Control_vizual()
	    MoveJ Target_control1,v500,z100,Flansa_Cuplare\WObj:=wobj_control;
	    MoveJ Target_control2,v500,z100,Flansa_Cuplare\WObj:=wobj_control;
	    SetDO\SDelay:=0,DO_deschide_cutie,0;
        TPWrite "Sistem de protectie ATI închis";
	    MoveJ Target_control3,v1000,z100,Flansa_Cuplare\WObj:=wobj_control;
	    MoveJ Target_control4,v1000,z50,Flansa_Cuplare\WObj:=wobj_control;
	    MoveJ Target_control5,v1000,z50,Flansa_Cuplare\WObj:=wobj_control;
	    MoveL Target_control6,v1000,z50,Flansa_Cuplare\WObj:=wobj_control;
	    MoveL Target_control7,v1000,z100,Flansa_Cuplare\WObj:=wobj_control;
	    MoveL Target_control8,v1000,z30,Flansa_Cuplare\WObj:=wobj_control;
	    MoveJ Target_control9,v1000,z30,Flansa_Cuplare\WObj:=wobj_control;
	    MoveJ Target_control10,v1000,z30,Flansa_Cuplare\WObj:=wobj_control;
	    MoveL Target_control11,v1000,z30,Flansa_Cuplare\WObj:=wobj_control;
	    MoveJ Target_control12,v1000,z30,Flansa_Cuplare\WObj:=wobj_control;
	    MoveL Target_control13,v1000,z30,Flansa_Cuplare\WObj:=wobj_control;
	    MoveL Target_control14,v1000,z30,Flansa_Cuplare\WObj:=wobj_control;
	    MoveL Target_control15,v1000,z30,Flansa_Cuplare\WObj:=wobj_control;
	    MoveJ Target_control16,v1000,z20,Flansa_Cuplare\WObj:=wobj_control;
	    MoveJ Target_control17,v1000,z30,Flansa_Cuplare\WObj:=wobj_control;
	    MoveL Target_control18,v1000,z30,Flansa_Cuplare\WObj:=wobj_control;
	    MoveJ Target_control19,v1000,z30,Flansa_Cuplare\WObj:=wobj_control;
	    MoveJ Target_control20,v1000,z30,Flansa_Cuplare\WObj:=wobj_control;
	    MoveL Target_control21,v1000,z30,Flansa_Cuplare\WObj:=wobj_control;
	    MoveJ Target_control22,v1000,z30,Flansa_Cuplare\WObj:=wobj_control;
	    MoveJ Target_control23,v1000,z30,Flansa_Cuplare\WObj:=wobj_control;
	    MoveL Target_control24,v1000,z30,Flansa_Cuplare\WObj:=wobj_control;
	    MoveJ Target_control25,v1000,z30,Flansa_Cuplare\WObj:=wobj_control;
	    MoveJ Target_control26,v1000,z30,Flansa_Cuplare\WObj:=wobj_control;
	    Path6_Cuplare_V;
	ENDPROC
    PROC Path6_Cuplare_V()
	    MoveJ Target_cuplare_V1,v400,z30,Flansa_Cuplare\WObj:=wobj_evacuare;
	    MoveJ Target_cuplare_V2,v400,z30,Tooldata_TCP_VAC\WObj:=wobj_evacuare;
	    WaitTime\InPos,0.5;
	    SetDO\SDelay:=1,do_cupleaza_V,1;
        TPWrite "Efector V cuplat";
	    WaitTime\InPos,1;
	    MoveJ Target_cuplare_V3,v400,z30,Tooldata_TCP_VAC\WObj:=wobj_evacuare;
	    MoveJ Target_cuplare_V4,v400,z30,Tooldata_TCP_VAC\WObj:=wobj_evacuare;
	    MoveJ Target_cuplare_V5,v1000,z30,Tooldata_TCP_VAC\WObj:=wobj_evacuare;
	    Path7_Evacuare_piesa;
	ENDPROC
	PROC Path7_Evacuare_piesa()
        TPWrite "Efectuare proces de evacuare a piesei debavurate";
	    MoveJ Target_evacuare1,v1000,z30,Tooldata_TCP_VAC\WObj:=wobj_evacuare;
	    MoveJ Target_evacuare2,v1000,z10,Tooldata_TCP_VAC\WObj:=wobj_evacuare;
	    MoveL Target_evacuare3,v300,z10,Tooldata_TCP_VAC\WObj:=wobj_evacuare;
	    WaitTime\InPos,1;
	    SetDO\SDelay:=0.5,DO_S4_Sistem_fixare,0;
	    SetDO\SDelay:=1,DO_S7_piesa_efector_V,1;
        TPWrite "Piesa debavurata preluata din sistemul de fixare";
	    WaitTime\InPos,1;
	    MoveL Target_evacuare4,v300,z10,Tooldata_TCP_VAC\WObj:=wobj_evacuare;
	    MoveJ Target_evacuare5,v1000,z30,Tooldata_TCP_VAC\WObj:=wobj_evacuare;
	    MoveJ Target_evacuare6,v1000,z30,Tooldata_TCP_VAC\WObj:=wobj_evacuare;
	    MoveJ Target_evacuare7,v1000,z30,Tooldata_TCP_VAC\WObj:=wobj_evacuare;
	    MoveJ Target_evacuare8,v1000,z30,Tooldata_TCP_VAC\WObj:=wobj_evacuare;
	    MoveJ Target_evacuare9,v1000,z30,Tooldata_TCP_VAC\WObj:=wobj_evacuare;
	    MoveJ Target_evacuare10,v1000,z30,Tooldata_TCP_VAC\WObj:=wobj_evacuare;
	    MoveJ Target_evacuare11,v300,z30,Tooldata_TCP_VAC\WObj:=wobj_evacuare;
	    WaitTime\InPos,1;
	    SetDO\SDelay:=1,DO_S7_piesa_efector_V,0;
        TPWrite "Piesa a fost depusa pe conveiorul de iesire";
	    SetDO\SDelay:=2,DO_piesa_gata,1;
	    WaitTime\InPos,1;
	    MoveJ Target_evacuare10,v300,z30,Tooldata_TCP_VAC\WObj:=wobj_evacuare;
	    MoveJ Target_evacuare12,v500,z100,Flansa_Cuplare\WObj:=wobj_alimentare;

        Incr pCounter;
        !Clear pCounter;
         TPWrite "Numarul de piese debavurate este:" \Num:=pCounter;
		Home;
	ENDPROC
ENDMODULE
